FUNCTION ARR08B_TO_BYTE
  (* Standard: 61499-1; Description: Copyright (c) 2024 franz This program and the accompanying materials are made available under the terms of the Eclipse Public License 2.0 which is available at https://www.eclipse.org/legal/epl-2.0/ SPDX-License-Identifier: EPL-2.0 *)
  (* Version 1.0, 2024-02-22, franz *)
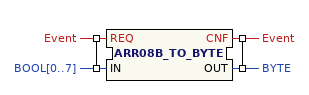
  EVENT_INPUT
    REQ WITH IN; (* Normal Execution Request *)
  END_EVENT
  EVENT_OUTPUT
    CNF WITH OUT; (* Execution Confirmation *)
  END_EVENT
  VAR_INPUT
    IN : ARRAY [0..7] OF BOOL; (* ARR08B Input *)
  END_VAR
  VAR_OUTPUT
    OUT : BYTE; (* BYTE Output *)
  END_VAR
  BODY IN ST:
FUNCTION ARR08B_TO_BYTE

VAR_INPUT
	IN : ARRAY[0..7] OF BOOL;    // ARR08B Input
END_VAR

VAR_OUTPUT
	OUT : BYTE;    // BYTE Output
END_VAR

(* this Function extracts the 8 Bits from a byte *)
OUT.0 := IN[0];
OUT.1 := IN[1];
OUT.2 := IN[2];
OUT.3 := IN[3];
OUT.4 := IN[4];
OUT.5 := IN[5];
OUT.6 := IN[6];
OUT.7 := IN[7];

END_FUNCTION
  END_BODY
END_FUNCTION
